FUNCTION_BLOCK FB_PWM_Output
(*
	Converts a real unit value (e.g., volts) to the integer needed for a PWM output terminal.
	2022-04-26 Maarten Thomas-Bosum
*)

// The following was copied from FB_AnalogOutput so the variables need to be updated according
// to the specifications of the EL2502 PWM Output terminal.

VAR_INPUT
	// The real value to send to the output
	fReal: LREAL;
	// The maximum allowed real value for the connected hardware
	fSafeMax: LREAL;
	// The minimum allowed real value for the connected hardware
	fSafeMin: LREAL;
	// The number of bits correlated with the terminal's max output. This is not necessarily the resolution parameter.
	iTermBits: UINT;
	// The fReal value correlated with the terminal's max output
	fTermMax: LREAL;
	// The fReal value correlated with the terminal's min output
	fTermMin: LREAL;
END_VAR
VAR_OUTPUT
	// Connect this output to the terminal
	iRaw AT %Q*: INT;
END_VAR
VAR
	fScale: LREAL;
END_VAR

// Set the scaling from real to raw
IF fScale = 0 AND fTermMax > fTermMin THEN
	fScale := (EXPT(2, iTermBits) - 1) / (fTermMax - fTermMin);
END_IF

// Adjust real value to be within the limits
fReal := MIN(fReal, fSafeMax, fTermMax);
fReal := MAX(fReal, fSafeMin, fTermMin);

// Scale the output accordingly
iRaw := LREAL_TO_INT((fReal - fTermMin) * fScale);

END_FUNCTION_BLOCK

(* stored: Version 1.1.0.1, ProductVersion 3.1.4022.18
   POU FB_PWM_Output: Id {563ecf95-0183-4061-b981-aa77c1abbdf1}, SpecialFunc None *)
